SUBAPPLICATION AX_2_TO_3 (* Konvertierung von 2 auf 3 AX-Adapter Signale *)
  (* Standard: 61499-2; Description: Copyright (c) 2026 HR Agrartechnik GmbH This program and the accompanying materials are made available under the terms of the Eclipse Public License 2.0 which is available at https://www.eclipse.org/legal/epl-2.0/ SPDX-License-Identifier: EPL-2.0 *)
  (* Version 1.0, 2026-04-19, Franz Höpfinger, HR Agrartechnik GmbH *)
  PACKAGE MyLib::sys;
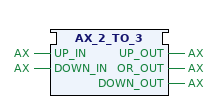
  SOCKETS
    UP_IN : adapter::types::unidirectional::AX;
    DOWN_IN : adapter::types::unidirectional::AX;
  END_SOCKETS
  PLUGS
    UP_OUT : adapter::types::unidirectional::AX;
    OR_OUT : adapter::types::unidirectional::AX;
    DOWN_OUT : adapter::types::unidirectional::AX;
  END_PLUGS
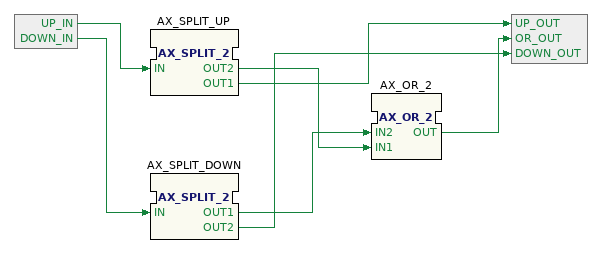
  FBS
    AX_SPLIT_DOWN : adapter::events::unidirectional::AX_SPLIT_2;
    AX_SPLIT_UP : adapter::events::unidirectional::AX_SPLIT_2;
    AX_OR_2 : adapter::booleanOperators::AX_OR_2;
  END_FBS
  ADAPTER_CONNECTIONS
    AX_SPLIT_DOWN.OUT1 TO AX_OR_2.IN2;
    AX_SPLIT_UP.OUT2 TO AX_OR_2.IN1;
    DOWN_IN TO AX_SPLIT_DOWN.IN;
    AX_SPLIT_DOWN.OUT2 TO DOWN_OUT;
    UP_IN TO AX_SPLIT_UP.IN;
    AX_SPLIT_UP.OUT1 TO UP_OUT;
    AX_OR_2.OUT TO OR_OUT;
  END_CONNECTIONS
END_SUBAPPLICATION
